{attribute 'pack_mode' := '1'}
TYPE ST_Complex_6 :
STRUCT
	a : INT := 42;
	b : DINT := 43;
	c : REAL := 42.42;
	d : LREAL := 42.42;
	e : INT := 44;
	f : BOOL := TRUE;
END_STRUCT
END_TYPE

(* stored: Version 1.1.0.1
   DUT ST_Complex_6: Id {186de150-16d1-45b8-89d2-7f4e8370c540} *)
